// TwinCAT 3 PLC project Plc_1
// ProgramVersion: 3.1.4024.0
// libraries:
//   Tc2_MC2, * (Beckhoff Automation GmbH)
//   Tc2_Standard, * (Beckhoff Automation GmbH)
//   Tc2_System, * (Beckhoff Automation GmbH)
//   Tc3_Module, * (Beckhoff Automation GmbH)
// project tree:
//   / PlcTask.TcTTO
//   POUs/ deneme.TcPOU, FB_ReversingSequence.TcPOU, MAIN.TcPOU
// real-time tasks:
//   TASK PlcTask: cycle T#10ms, priority 20, ADS port 350
// motion (NC):
//   TASK NC-Task 1 SAF: cycle T#2ms, priority 4, ADS port 501
//   TASK NC-Task 1 SVB: cycle T#10ms, priority 8, ADS port 511
//   AXIS Axis 1 (id 1)
//     OtherSettings: AllowMotionCmdToSlave=true
//     encoder EncType=1
//     drive DrvType=5
//       Analog: TorqueSetpointScale=10, ScaleFactorActTorque=0.1
//       TimeComp: TaskDelayCycles=1
//     controller CtrType=1
//       CtrPara: PriorControlFactor=1
//         Observer: BandWidth=20
//   AXIS Axis 2 (id 2)
//     OtherSettings: AllowMotionCmdToSlave=true
//     encoder EncType=1
//     drive DrvType=5
//       Analog: TorqueSetpointScale=10, ScaleFactorActTorque=0.1
//       TimeComp: TaskDelayCycles=1
//     controller CtrType=1
//       CtrPara: PriorControlFactor=1
//         Observer: BandWidth=20
// variable links:
//   Plc-1/Plc-1 Instance <-> NC-Task 1 SAF/Axes/Axis 1
//     PlcTask Inputs/MAIN.axis_1.NcToPlc <-> Outputs/ToPlc
//     PlcTask Outputs/MAIN.axis_1.PlcToNc <-> Inputs/FromPlc

CONFIGURATION Plc_1
    RESOURCE PLC ON TwinCAT3
        TASK PlcTask(INTERVAL := T#10ms, PRIORITY := 20);
        PROGRAM MAIN WITH PlcTask : MAIN;
    END_RESOURCE
END_CONFIGURATION

// ---- POUs/MAIN.TcPOU
PROGRAM MAIN
VAR
	axis_1 			:AXIS_REF;
	axis_2			:AXIS_REF;
	fbEnable		:MC_Power;
	bEnable			:BOOL;
	fbAbsolute		:MC_MoveAbsolute;
	bAbsolute		:BOOL;
	fbRelative		:MC_MoveRelative;
	bRelative		:BOOL;
//Axis: INT; otomatik oluşturdu neden integer?
	
	
	
	fbReversingSequence: FB_ReversingSequence;
	fPosition1: LREAL;
	fPosition2: LREAL;
	fVelocity: LREAL;
	tDelay: TIME;
	bError: BOOL;
	sStatus: STRING;
	deneme: deneme;
END_VAR

(*fbEnable(
	Axis:= axis_1 , //eğer axis vermezsek hata alırız.
	Enable:=bEnable , 
	Enable_Positive:=bEnable , 
	Enable_Negative:= bEnable, 
	Override:= 100//sistemin ne kadar kullanılacağı ???
 );
fbAbsolute(
	Axis:=axis_1 , 
	Execute:= bAbsolute, 
	Position:= 1500, 
	Velocity:= 500);
	
fbRelative(

	Axis:=axis_1 , 
	Execute:= bRelative, 
	Distance:= 1000, 
	Velocity:=500 );	
	*)
	
	(*fbReversingSequence(
	bEnable:=bEnable , 
	fPosition1:=fPosition1 , 
	fPosition2:= fPosition2, 
	fVelocity:= fVelocity, 
	tDelay:= tDelay, 
	bError=> bError, 
	sStatus=>sStatus , 
	Axis:= axis_1);*)
	deneme(
	bEnable:=bEnable , 
	fPosition1:=fPosition1 , 
	fPosition2:=fPosition2 , 
	fVelocity:=fVelocity , 
	tDelay:=tDelay , 
	bError=>bError , 
	sStatus=>sStatus , 
	Axis:=axis_1 , 
	Axis2:=axis_2 );

END_PROGRAM

// ---- POUs/FB_ReversingSequence.TcPOU
FUNCTION_BLOCK FB_ReversingSequence
VAR_INPUT
	bEnable 		: BOOL;
	fPosition1 		: LREAL; //pozisyon tiplerimiz LREAL'dir.
	fPosition2 		: LREAL;
	fVelocity		: LREAL;
	tDelay 			: TIME;
END_VAR
VAR_OUTPUT
	bError 			: BOOL;
	sStatus 		: STRING;
END_VAR
VAR
	fbPower			: MC_Power;
	fbMove			: MC_MoveAbsolute;
	nState			: INT;
	fbTimer 		: TON;
END_VAR
VAR_IN_OUT
	Axis		:AXIS_REF;
//Axisler VAR_IN_OUT değişkenleridir sadece onun içinde tanımlanır!!.
END_VAR


fbPower(
	Axis:=Axis , 
	Enable:=TRUE , 
	Enable_Positive:=TRUE, 
	Enable_Negative:=TRUE , 
	Override:=100  );

	fbMove(
	Axis:=Axis , 
	Velocity:=  fVelocity);
	
	Axis.ReadStatus();
	
	fbTimer(PT:= tDelay);
CASE nState OF
	0: //eksenin Enable state'i
		bError 		:=FALSE;
		sStatus 	:='Beklemede';
		IF bEnable AND Axis.Status.Operational THEN
			nState :=10;
			ELSIF NOT Axis.Status.Operational THEN
				nState :=900;
				sStatus :='Enable değil';
		END_IF
		
	10: //Execute state'i
	fbMove.Position :=fPosition1;
	fbMove.Execute := TRUE;
	IF Axis.Status.Moving THEN
		sStatus 	:='1. noktaya Hareket ediyor';
		nState :=20;
		ELSIF Axis.Status.Error OR fbMove.Error THEN
			sStatus 	:='1. noktaya giderken hataya geçti';
			nstate :=900;
	END_IF
	
	20://hareket kontrol state'i
		IF fbMove.Done THEN
			nState := 30;
			fbMove.Execute :=FALSE;
//2. hareketi de yapmak için false dedik.	
			
		END_IF
		
	30:
		
		fbTimer.IN:=TRUE;
		sStatus:='1. Noktada bekliyor.';
		
		IF(fbTimer.Q) THEN
			fbTimer.IN:=FALSE;
			nState:=40;
		END_IF
		
	40://2. hareket.
		fbMove.Position :=fPosition2;
		fbMove.Execute := TRUE;
		IF Axis.Status.Moving THEN
			sStatus 	:='2. noktaya Hareket ediyor';
			nState :=50;
		ELSIF Axis.Status.Error OR fbMove.Error THEN
			sStatus 	:='2. noktaya giderken hataya geçti';
			nstate :=900;
		END_IF
		
	50:
		IF fbMove.Done THEN
			nState := 60;
			fbMove.Execute :=FALSE;
		END_IF
		
	60: 
		fbTimer.IN:=TRUE;
		sStatus:='2. Noktada bekliyor.';
		
		IF(fbTimer.Q) THEN
			fbTimer.IN:=FALSE;
			nState:=0;
		END_IF
		
		
	900:
		bError := TRUE;
		IF NOT bEnable THEN
			fbTimer(IN:=FALSE);
			nState:=0;
		END_IF
		
END_CASE

END_FUNCTION_BLOCK

// ---- POUs/deneme.TcPOU
FUNCTION_BLOCK deneme
VAR_INPUT//girilecek değerler
	bEnable			: BOOL;
	fPosition1		: LREAL;
	fPosition2		: LREAL;
	fVelocity		: LREAL;
	tDelay 			: TIME;
END_VAR
VAR_OUTPUT
	bError			: BOOL;
	sStatus 		: STRING;
END_VAR
VAR//kullanıcının görmesine gerek yok!
	fbPower 		: MC_Power;
	fbPower2		: MC_Power;
	fbMove 			: MC_MoveAbsolute;
	fbMove2			: MC_MoveAbsolute;
	nState 			: INT;
	fbTimer 		: TON;
END_VAR

VAR_IN_OUT 
	Axis 		:AXIS_REF;
	Axis2		:AXIS_REF;
END_VAR

fbPower2(
	Axis:= Axis2, 
	Enable:= TRUE, 
	Enable_Positive:= TRUE, 
	Enable_Negative:= TRUE, 
	Override:=  100);
fbMove2(
	Axis:= Axis2, 
	Velocity:=fVelocity , 
);
fbPower(
	Axis:= Axis, 
	Enable:= TRUE , 
	Enable_Positive:= TRUE, 
	Enable_Negative:= TRUE, 
	Override:=100);
	
	fbMove(
	Axis:= Axis, 
	Velocity:= fVelocity);
	
	Axis.ReadStatus();
	Axis2.ReadStatus();
	
	fbTimer(PT:= tDelay);
	CASE nState OF
	0://eksen enable state
			bError:=FALSE;
			sStatus :='Beklemede';
			IF bEnable AND Axis.Status.Operational AND Axis2.Status.Operational THEN
				nState :=10;
				ELSIF NOT  Axis.Status.Operational OR Axis2.Status.Operational THEN
					nState :=900;
					sStatus :='Enable değil';
			END_IF
			
	10://Execute state'i.
		fbMove.Position:=fPosition1;
		fbMove2.Position:=fPosition2;
		fbMove.Execute:=TRUE;
		IF Axis.Status.Moving AND Axis2.Status.Moving THEN
			sStatus 	:='Eksenler ilk noktaya Hareket ediyor.';
			nState:=20;
			ELSIF Axis.Status.Error OR fbMove.Error OR Axis2.Status.Error OR fbMove2.Error  THEN
				sStatus :='1. noktaya giderken hataya geçti';
				nState :=900;
		END_IF
			
	20://hareket kontrol state'i.
		IF fbMove.Done AND fbMove2.Done THEN
			sStatus 		:='1. Noktaya vardı';
			nState 			:=30;
			fbMove.Execute:=FALSE;//2. hareket için false'a çektik.
			fbMove2.Execute:=FALSE;
			
		END_IF
		
	30: //timer state
		fbTimer.IN:= TRUE;
		sStatus:='1. Noktada bekliyor.';
		IF(fbTimer.Q) THEN
			fbTimer.IN:=FALSE;
			nState :=40;
			
		END_IF
	40://2. noktaya hareket.
		fbMove2.Position:=fPosition2;
		fbMove.Position:=fPosition1;
		fbMove.Execute:=TRUE;
		fbMove2.Execute:=TRUE;
		IF Axis.Status.Moving AND Axis2.Status.Moving THEN
			sStatus :='2. noktaya hareket ediyor';
			nState := 50;
		ELSIF  Axis.Status.Error OR fbMove.Error OR Axis2.Status.Error OR fbMove2.Error THEN
			sStatus :='2. noktaya geçerken hataya geçti';
			nState :=900;
		END_IF
	50:
		IF fbMove.Done AND fbMove2.Done THEN
			sStatus :='2. noktaya vardı.';
			nstate :=60;
			fbMove.Execute:=FALSE;
			
		END_IF
	60:
		fbTimer.IN:=TRUE;
		sStatus :='2. noktada bekliyor';
		IF fbTimer.Q THEN
			fbTimer.IN:=FALSE;			
			nState :=0;
		END_IF
	900:
		bError := TRUE;
		IF NOT bEnable THEN
			fbTimer(IN:=FALSE);
			nState:=0;
		END_IF
		
	END_CASE

END_FUNCTION_BLOCK
